// TIA Portal V20 export
TYPE "typeEm6MonitoringSoftCam"
// stored: Access Published, Namespace Unit1
   STRUCT
      VisionUnit { ExternalWritable := 'False'} : "LER_typeSoftCamRelation";
   END_STRUCT;
   // // VisionUnit.posistion0 : HomePos
   // // VisionUnit.posistion1 : VisionPos
END_TYPE
